PROGRAM NstBkgrdLsSerialCom
VAR_INPUT
	Config : NstConfig;
END_VAR
VAR
END_VAR

// AttenuationFilterConfigs
IF Config.AttenuationFilterConfigs.FW212CAttenuationFilterConfig.IsEnabled OR 
   Config.AttenuationFilterConfigs.ELL14kAttenuationFilterConfig.IsEnabled OR 
   Config.AttenuationFilterConfigs.ELL9AttenuationFilterConfig.IsEnabled THEN
	BkgrdSerialAttenuation();	
END_IF

// LaserConfigs
IF Config.LaserConfigs.SMD12LaserConfig.IsEnabled OR 
   Config.LaserConfigs.Piano450LaserConfig.IsEnabled THEN
	BkgrdSerialLaser();
END_IF

END_PROGRAM

(* stored: Version 1.1.0.1, ProductVersion 3.1.4024.12
   POU NstBkgrdLsSerialCom: Id {b1cfc9e4-3d08-4cd4-9bde-220900b9077a}, SpecialFunc None *)
